// TIA Portal V16 export
// export: Created 2019-09-22T13:16:38.027184Z, ExportSetting WithDefaults, DisplayName Totally Integrated Automation Portal, DisplayVersion V16, DisplayName TIA Portal Version Control Interface, DisplayVersion V16, DisplayName TIA Portal Openness, DisplayVersion V16, DisplayName STEP 7 Professional, DisplayVersion V16, DisplayName SIMATIC Energy Suite, DisplayVersion V16, DisplayName STEP 7 Safety, DisplayVersion V16, DisplayName WinCC Professional, DisplayVersion V16, DisplayName SIMATIC Visualization Architect, DisplayVersion V16
FUNCTION_BLOCK "LiftSim"   // FB140, FBD
{ S7_Optimized_Access := 'TRUE' }
VERSION : 0.1
// stored: AutoNumber true, IsIECCheckEnabled false, IsRetainMemResEnabled false, MemoryReserve 100, SetENOAutomatically false, UDAEnableTagReadback false
   VAR
      instRisTrigLift1 { S7_SetPoint := 'True'} : R_TRIG;
      instRisTrigLift2 { S7_SetPoint := 'True'} : R_TRIG;
      risTrigLift1 : Bool;
      risTrigLift2 : Bool;
      instFrequency { S7_SetPoint := 'True'} : "LGF_Frequency";
      instRisTrigClock { S7_SetPoint := 'True'} : R_TRIG;
      statRisTrigClock : Bool;
      statClock10Hz : Bool;
   END_VAR
   VAR CONSTANT
      POS_STOPPER_1 : Int := 50;   // Position case stopper 1
      POS_STOPPER_2 : Int := 74;   // Position case stopper 2
      POS_STOPPER_3 : Int := 100;   // Position case stopper 3
      POS_LIFT_TOP : Int := 60;   // Position of lift at top
      POS_LIFT_BOTTOM : Int := 0;   // Position of lift at bottom
   END_VAR
BEGIN

REGION Network 1
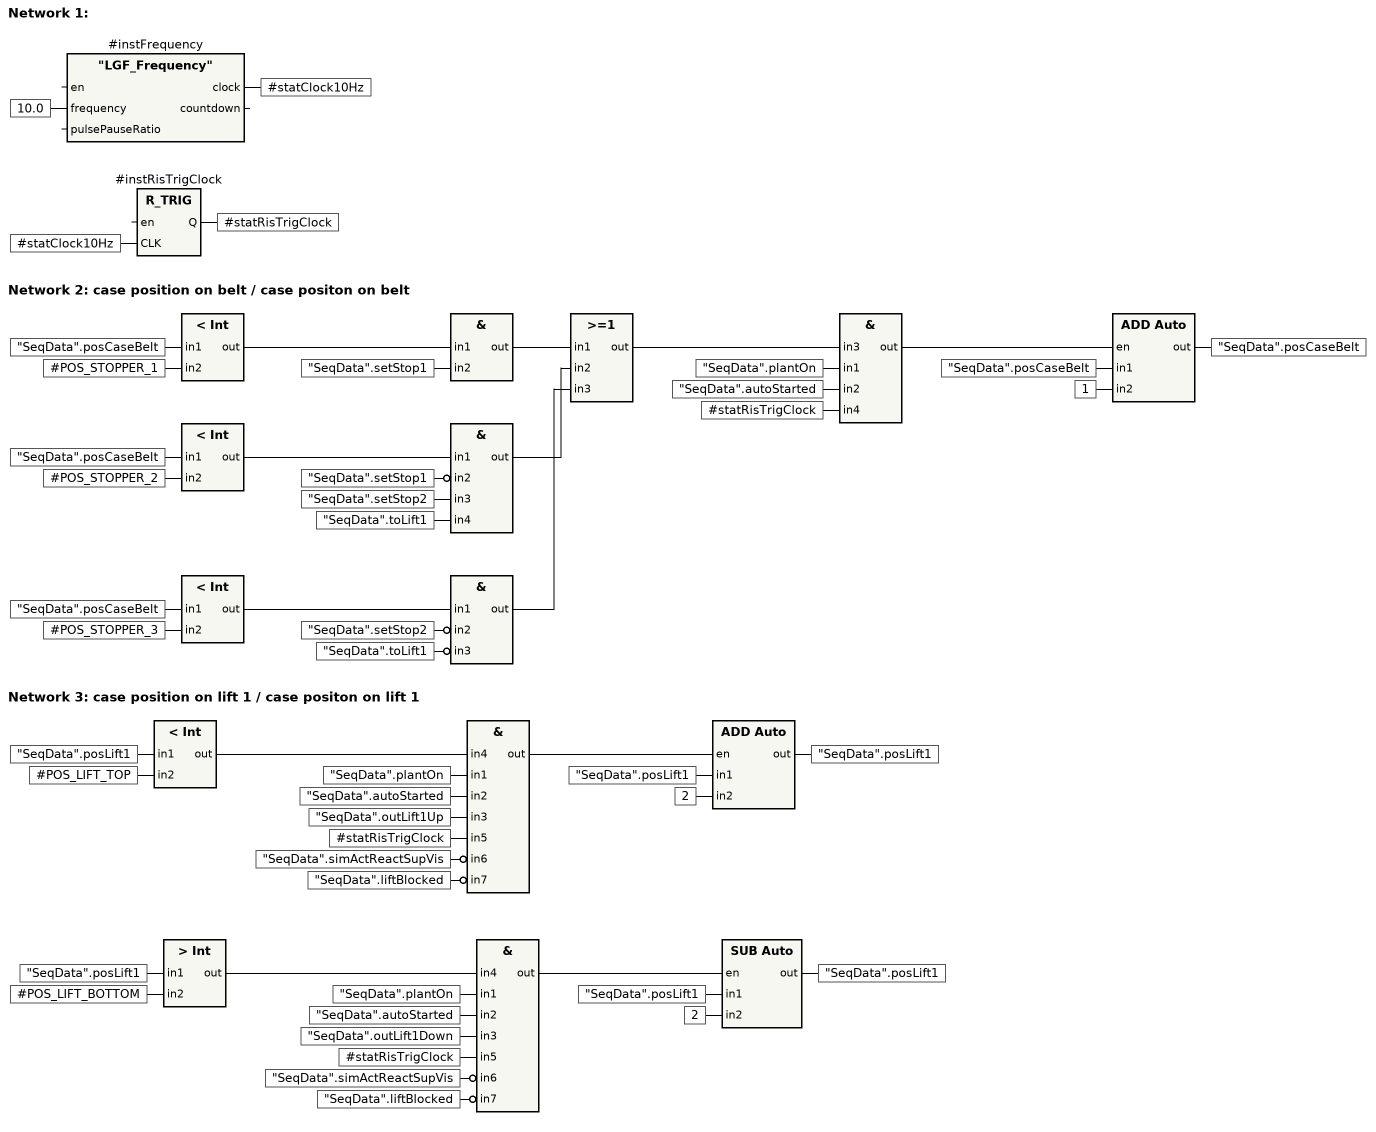
   #instFrequency(frequency := 10.0, clock => #statClock10Hz);   // "LGF_Frequency"
   #instRisTrigClock(CLK := #statClock10Hz, Q => #statRisTrigClock);   // R_TRIG
END_REGION

REGION Network 2: case position on belt / case positon on belt
   IF ((("SeqData".posCaseBelt < #POS_STOPPER_1) AND "SeqData".setStop1) OR (("SeqData".posCaseBelt < #POS_STOPPER_2) AND NOT "SeqData".setStop1 AND "SeqData".setStop2 AND "SeqData".toLift1) OR (("SeqData".posCaseBelt < #POS_STOPPER_3) AND NOT "SeqData".setStop2 AND NOT "SeqData".toLift1)) AND "SeqData".plantOn AND "SeqData".autoStarted AND #statRisTrigClock THEN
       "SeqData".posCaseBelt := "SeqData".posCaseBelt + 1;
   END_IF;
END_REGION

REGION Network 3: case position on lift 1 / case positon on lift 1
   IF ("SeqData".posLift1 < #POS_LIFT_TOP) AND "SeqData".plantOn AND "SeqData".autoStarted AND "SeqData".outLift1Up AND #statRisTrigClock AND NOT "SeqData".simActReactSupVis AND NOT "SeqData".liftBlocked THEN
       "SeqData".posLift1 := "SeqData".posLift1 + 2;
   END_IF;
   IF ("SeqData".posLift1 > #POS_LIFT_BOTTOM) AND "SeqData".plantOn AND "SeqData".autoStarted AND "SeqData".outLift1Down AND #statRisTrigClock AND NOT "SeqData".simActReactSupVis AND NOT "SeqData".liftBlocked THEN
       "SeqData".posLift1 := "SeqData".posLift1 - 2;
   END_IF;
END_REGION

REGION Network 4: case position on lift 2 / case positon on lift 2
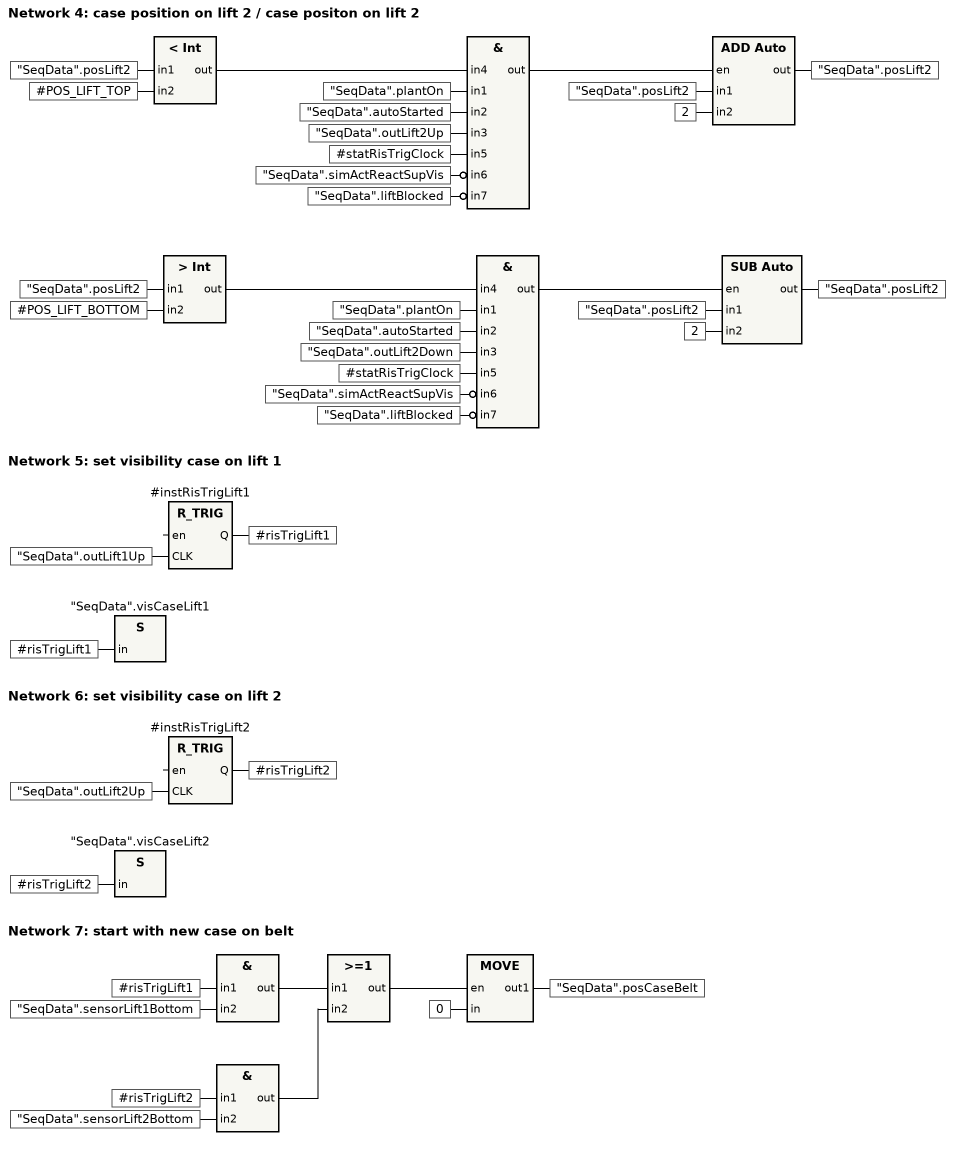
   IF ("SeqData".posLift2 < #POS_LIFT_TOP) AND "SeqData".plantOn AND "SeqData".autoStarted AND "SeqData".outLift2Up AND #statRisTrigClock AND NOT "SeqData".simActReactSupVis AND NOT "SeqData".liftBlocked THEN
       "SeqData".posLift2 := "SeqData".posLift2 + 2;
   END_IF;
   IF ("SeqData".posLift2 > #POS_LIFT_BOTTOM) AND "SeqData".plantOn AND "SeqData".autoStarted AND "SeqData".outLift2Down AND #statRisTrigClock AND NOT "SeqData".simActReactSupVis AND NOT "SeqData".liftBlocked THEN
       "SeqData".posLift2 := "SeqData".posLift2 - 2;
   END_IF;
END_REGION

REGION Network 5: set visibility case on lift 1
   #instRisTrigLift1(CLK := "SeqData".outLift1Up, Q => #risTrigLift1);   // R_TRIG
   IF #risTrigLift1 THEN "SeqData".visCaseLift1 := TRUE; END_IF;
END_REGION

REGION Network 6: set visibility case on lift 2
   #instRisTrigLift2(CLK := "SeqData".outLift2Up, Q => #risTrigLift2);   // R_TRIG
   IF #risTrigLift2 THEN "SeqData".visCaseLift2 := TRUE; END_IF;
END_REGION

REGION Network 7: start with new case on belt
   IF (#risTrigLift1 AND "SeqData".sensorLift1Bottom) OR (#risTrigLift2 AND "SeqData".sensorLift2Bottom) THEN
       "SeqData".posCaseBelt := 0;
   END_IF;
END_REGION

REGION Network 8: check, if new case
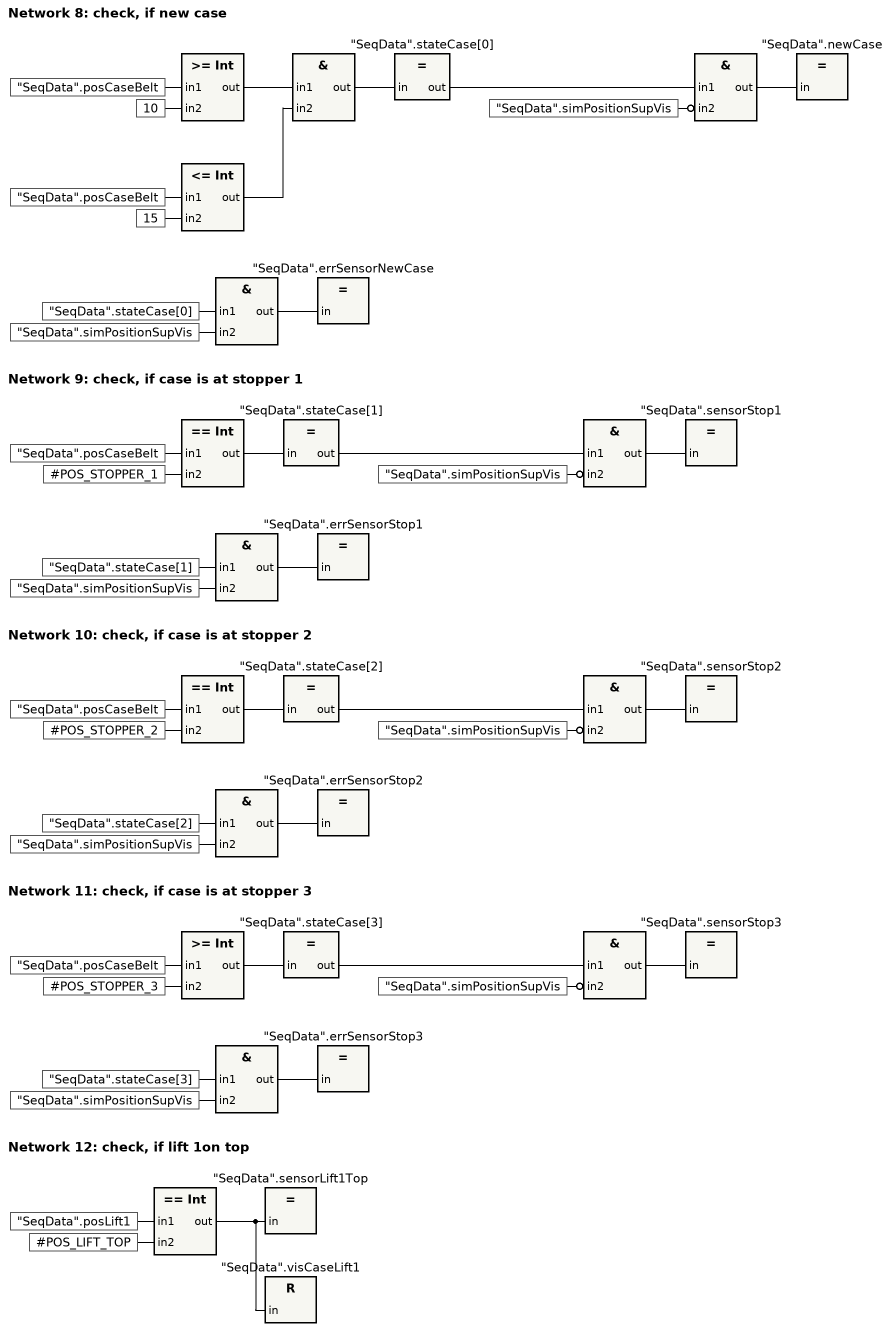
   "SeqData".stateCase[0] := ("SeqData".posCaseBelt >= 10) AND ("SeqData".posCaseBelt <= 15);
   "SeqData".newCase := ("SeqData".posCaseBelt >= 10) AND ("SeqData".posCaseBelt <= 15) AND NOT "SeqData".simPositionSupVis;
   "SeqData".errSensorNewCase := "SeqData".stateCase[0] AND "SeqData".simPositionSupVis;
END_REGION

REGION Network 9: check, if case is at stopper 1
   "SeqData".stateCase[1] := "SeqData".posCaseBelt = #POS_STOPPER_1;
   "SeqData".sensorStop1 := ("SeqData".posCaseBelt = #POS_STOPPER_1) AND NOT "SeqData".simPositionSupVis;
   "SeqData".errSensorStop1 := "SeqData".stateCase[1] AND "SeqData".simPositionSupVis;
END_REGION

REGION Network 10: check, if case is at stopper 2
   "SeqData".stateCase[2] := "SeqData".posCaseBelt = #POS_STOPPER_2;
   "SeqData".sensorStop2 := ("SeqData".posCaseBelt = #POS_STOPPER_2) AND NOT "SeqData".simPositionSupVis;
   "SeqData".errSensorStop2 := "SeqData".stateCase[2] AND "SeqData".simPositionSupVis;
END_REGION

REGION Network 11: check, if case is at stopper 3
   "SeqData".stateCase[3] := "SeqData".posCaseBelt >= #POS_STOPPER_3;
   "SeqData".sensorStop3 := ("SeqData".posCaseBelt >= #POS_STOPPER_3) AND NOT "SeqData".simPositionSupVis;
   "SeqData".errSensorStop3 := "SeqData".stateCase[3] AND "SeqData".simPositionSupVis;
END_REGION

REGION Network 12: check, if lift 1on top
   "SeqData".sensorLift1Top := "SeqData".posLift1 = #POS_LIFT_TOP;
   IF "SeqData".sensorLift1Top THEN "SeqData".visCaseLift1 := FALSE; END_IF;
END_REGION

REGION Network 13: check, if lift 2 on top
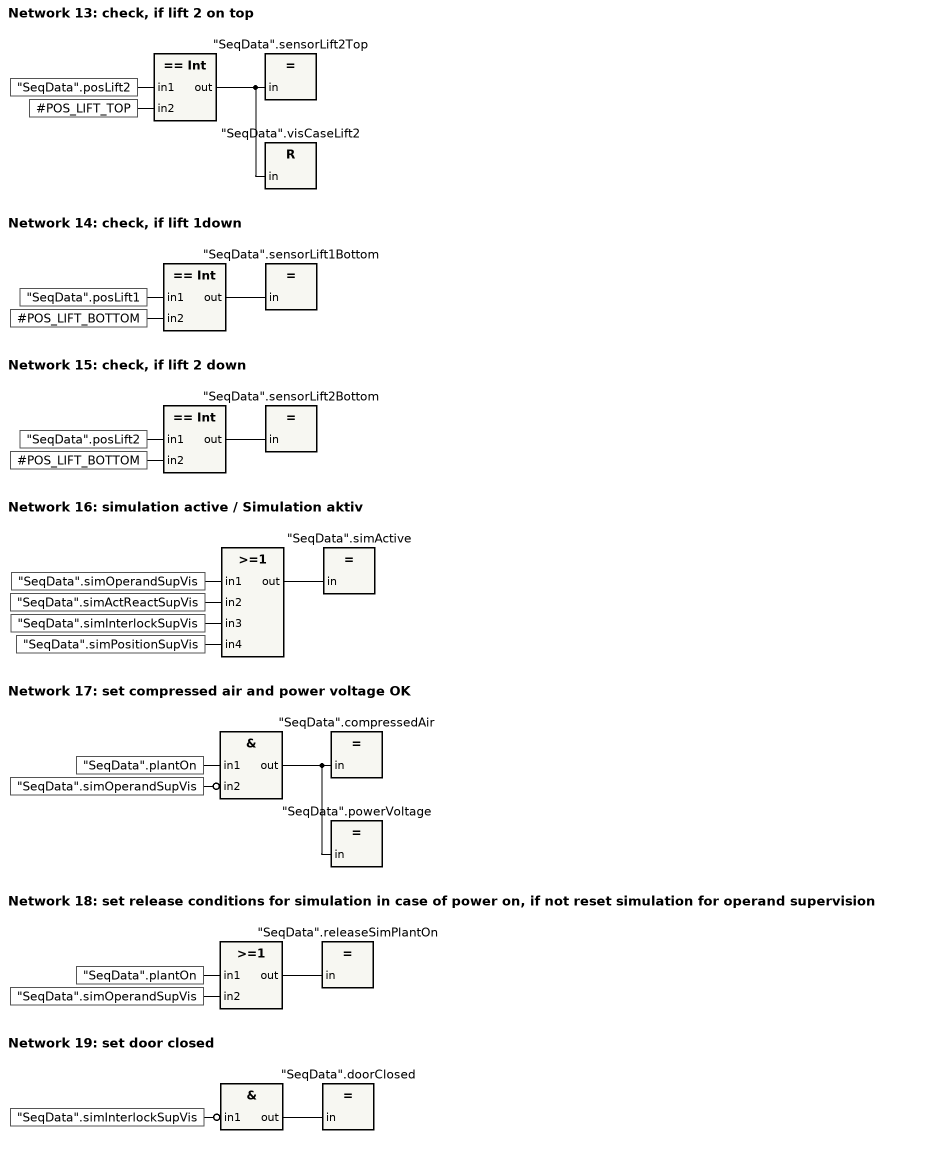
   "SeqData".sensorLift2Top := "SeqData".posLift2 = #POS_LIFT_TOP;
   IF "SeqData".sensorLift2Top THEN "SeqData".visCaseLift2 := FALSE; END_IF;
END_REGION

REGION Network 14: check, if lift 1down
   "SeqData".sensorLift1Bottom := "SeqData".posLift1 = #POS_LIFT_BOTTOM;
END_REGION

REGION Network 15: check, if lift 2 down
   "SeqData".sensorLift2Bottom := "SeqData".posLift2 = #POS_LIFT_BOTTOM;
END_REGION

REGION Network 16: simulation active / Simulation aktiv
   "SeqData".simActive := "SeqData".simOperandSupVis OR "SeqData".simActReactSupVis OR "SeqData".simInterlockSupVis OR "SeqData".simPositionSupVis;
END_REGION

REGION Network 17: set compressed air and power voltage OK
   "SeqData".compressedAir := "SeqData".plantOn AND NOT "SeqData".simOperandSupVis;
   "SeqData".powerVoltage := "SeqData".compressedAir;
END_REGION

REGION Network 18: set release conditions for simulation in case of power on, if not reset simulation for operand supervision
   "SeqData".releaseSimPlantOn := "SeqData".plantOn OR "SeqData".simOperandSupVis;
END_REGION

REGION Network 19: set door closed
   // Simulate the error that the door was openend / Fehlersimulation
   "SeqData".doorClosed := NOT "SeqData".simInterlockSupVis;
END_REGION
END_FUNCTION_BLOCK
